FUNCTION_BLOCK SimpleTestINC (* Template for an empty simple function block *)
  (* Standard: 61499-1; Description: Copyright (c) 2019 Jan Holzweber This program and the accompanying materials are made available under the terms of the Eclipse Public License 2.0 which is available at https://www.eclipse.org/legal/epl-2.0/ SPDX-License-Identifier: EPL-2.0 *)
  (* Version 1.0, 2019-06-11, Jan Holzweber *)
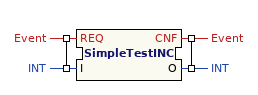
  EVENT_INPUT
    REQ WITH I; (* Normal Execution Request *)
  END_EVENT
  EVENT_OUTPUT
    CNF WITH O; (* Execution Confirmation *)
  END_EVENT
  VAR_INPUT
    I : INT;
  END_VAR
  VAR_OUTPUT
    O : INT;
  END_VAR
  ALGORITHM REQ IN ST:
O := I +1;
  END_ALGORITHM
END_FUNCTION_BLOCK
